# EPICS substitutions: xrmIocApp/Db/ch8.substitutions
file "ch.template"
{
	pattern {ch}
	{01}
	{02}
	{03}
	{04}
	{05}
	{06}
	{07}
	{08}
}
